INTERFACE I_TestResultLogger

METHOD PUBLIC LogTestSuiteResults
END_METHOD

METHOD ResetTestResultLogger
END_METHOD

END_INTERFACE

(* stored: Version 1.1.0.1, ProductVersion 3.1.4024.11
   Itf I_TestResultLogger: Id {fa75ee61-43fb-4767-8061-125a3a9e3424}
   Method LogTestSuiteResults: Id {033e8873-ad7a-489b-8ba9-f0de8a344939}
   Method ResetTestResultLogger: Id {0cecc36c-b023-434c-b61d-6002a0b2db3d} *)
